INTERFACE ITcoArguments

METHOD AddBool : ITcoArguments
VAR_INPUT
	Value		: BOOL;
END_VAR
END_METHOD

METHOD AddDecimal : ITcoArguments
VAR_INPUT
	Value	: DINT;
END_VAR
END_METHOD

METHOD AddFloat : ITcoArguments
VAR_INPUT
	Value	: LREAL;
END_VAR
END_METHOD

METHOD AddString : ITcoArguments
VAR_INPUT
	Value	: STRING(255);
END_VAR
END_METHOD

METHOD AddStruct : ITcoArguments
VAR_INPUT
	ioSIZE 		: UDINT;
	pVARIABLE 	: POINTER TO ULINT;
END_VAR
END_METHOD

METHOD Append : ITcoLogger
VAR_INPUT
END_VAR
END_METHOD

END_INTERFACE

(* stored: Version 1.1.0.1, ProductVersion 3.1.4024.9
   Itf ITcoArguments: Id {ba8c61a3-2b32-0265-3d0f-67adc21c68ec}
   Method AddBool: Id {76119336-76c3-0e1c-0027-3825da5a6dd7}
   Method AddDecimal: Id {32cc8609-26f4-08f2-301d-c69f08d6ed9a}
   Method AddFloat: Id {7edc0df8-d3b3-0cea-24f0-c71474b00bff}
   Method AddString: Id {c69ccdfa-d6bd-05a5-2320-b6dd9b22cf01}
   Method AddStruct: Id {b03ec0bd-06a4-0d16-0d03-e91004337e7f}
   Method Append: Id {b56d5192-7708-036c-2639-da473fcc2ea4} *)
